FUNCTION_BLOCK FB_PDER_TO_P (* Estimates underated PV power from derated PV power and deration factor. *)
  (* Standard: 61499-2; Description: Division by zero is avoided. *)
  (* Version 0.0, 2017-06-28, Marc Jakobi, HTW Berlin *)
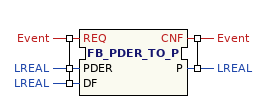
  EVENT_INPUT
    REQ WITH PDER, DF; (* Normal Execution Request *)
  END_EVENT
  EVENT_OUTPUT
    CNF WITH P; (* Execution Confirmation *)
  END_EVENT
  VAR_INPUT
    PDER : LREAL; (* Derated power *)
    DF : LREAL; (* Derating factor *)
  END_VAR
  VAR_OUTPUT
    P : LREAL; (* Non-derated power *)
  END_VAR
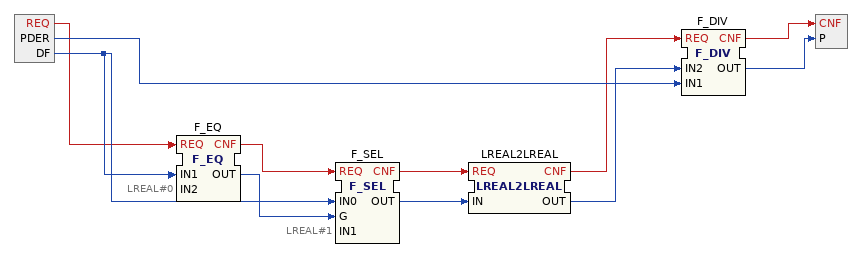
  FBS
    F_DIV : F_DIV;
    F_EQ : F_EQ(IN2 := LREAL#0);
    F_SEL : F_SEL(IN1 := LREAL#1);
    LREAL2LREAL : LREAL2LREAL;
  END_FBS
  EVENT_CONNECTIONS
    REQ TO F_EQ.REQ;
    F_EQ.CNF TO F_SEL.REQ;
    F_SEL.CNF TO LREAL2LREAL.REQ;
    LREAL2LREAL.CNF TO F_DIV.REQ;
    F_DIV.CNF TO CNF;
  END_CONNECTIONS
  DATA_CONNECTIONS
    DF TO F_EQ.IN1;
    DF TO F_SEL.IN0;
    F_EQ.OUT TO F_SEL.G;
    F_SEL.OUT TO LREAL2LREAL.IN;
    LREAL2LREAL.OUT TO F_DIV.IN2;
    PDER TO F_DIV.IN1;
    F_DIV.OUT TO P;
  END_CONNECTIONS
END_FUNCTION_BLOCK
